Fanuc KAREL source: RMCN_SEND.kl

PROGRAM T
%NOLOCKGROUP
VAR
 v0 : STRING[40]
 v1 : ARRAY[10] OF STRING[40]
 v2 : INTEGER
 v3 : INTEGER
BEGIN
 RMCN_SEND(v0, v1, v2, v3)
END T
